FUNCTION_BLOCK EL2872
VAR
	{attribute addProperty Name "WcState"}
	_wcState : WcStateBase;
	{attribute addProperty Name "Info data"}
	_infoData : InfoDataBase;
	_io : EL2xx9_Data;
END_VAR

PROPERTY IO : REFERENCE TO EL2xx9_Data
GET
IO REF= _io;
END_GET
END_PROPERTY

PROPERTY WcState : REFERENCE TO WcStateBase
GET
WcState REF= _wcState;
END_GET
END_PROPERTY

END_FUNCTION_BLOCK

(* stored: Version 1.1.0.1, ProductVersion 3.1.4024.9
   POU EL2872: Id {2d2e262f-747c-0ea6-2f72-84190a74e24a}, SpecialFunc None
   Property IO: Id {2fc8aa60-792d-0688-228d-224164a8ec22}
   Get Get: Id {b6a3a333-9fcf-04bd-3bfc-80f50468f4ee}
   Property WcState: Id {03848f57-4e84-078f-01b2-f200970594d0}
   Get Get: Id {2c936269-f70c-0c36-3089-54cf94207f5a} *)
